// TIA Portal V17 export
// export: Created 2023-02-23T17:15:49.9931985Z, ExportSetting WithDefaults, DisplayName Totally Integrated Automation Portal, DisplayVersion V17, DisplayName TIA Portal Openness, DisplayVersion V17, DisplayName TIA Portal Version Control Interface, DisplayVersion V17, DisplayName TIA Portal Test Suite Advanced, DisplayVersion V17, DisplayName STEP 7 Professional, DisplayVersion V17, DisplayName SIMATIC Energy Suite, DisplayVersion V17, DisplayName STEP 7 Safety, DisplayVersion V17, DisplayName WinCC Professional, DisplayVersion V17
DATA_BLOCK "MAN_ControlLine_DB_1"   // DB5
VERSION : 0.1
// stored: AutoNumber true, InstanceOfName MAN_ControlLine, InstanceOfType FB
"MAN_ControlLine"
   // VAR_INPUT
   //    ButtonStart : Bool;
   //    ButtonStop : Bool;
   //    ModeManual : Bool;
   //    ModeAuto : Bool;
   //    GlobalError : Bool;
   //    FirstScan : Bool;
   // END_VAR
   // VAR_OUTPUT
   //    StartLine : Bool;
   //    StopLine : Bool;
   //    AlarmSiren : Bool;
   // END_VAR
   // VAR
   //    s1 : Bool;
   //    s2 : Bool;
   //    s3 : Bool;
   //    s4 : Bool;
   //    P_ButtonStart_1 : Bool;
   //    P_ButtonStart_2 : Bool;
   //    IEC_Timer_0_Instance { ExternalAccessible := 'False'; ExternalVisible := 'False'; ExternalWritable := 'False'} : TP_TIME;
   //    Run { S7_SetPoint := 'True'} : Bool;
   //    N_Run : Bool;
   // END_VAR
BEGIN
END_DATA_BLOCK
